TYPE (* logiBUS_DI Struct *)
  (* Version 1.0, 2025-07-21, franz *)
  logiBUS_DI_Events_S : STRUCT
    EType : USINT := 255;
  END_STRUCT;
END_TYPE
